(* PLC project HdySimulator Functions library, Porcheson AuxBAse Framework 0.0 *)
(* stored: creationDateTime 2023-02-10T00:00:00, modificationDateTime 2026-02-10T00:00:00 *)

FUNCTION_BLOCK HDY_CreateSimAxis
  VAR_INPUT
    AXISTYPE : USINT;
    MAXVEL : REAL;
    MAXACC : REAL;
    MAXDEC : REAL;
  END_VAR
  VAR_OUTPUT
    AXISID : SINT;
    DONE : BOOL;
  END_VAR

						{{ extern void __mcl_cmd_createSimAxis(HDY_CREATESIMAXIS *data__);	__mcl_cmd_createSimAxis(data__);	 }}	
					
END_FUNCTION_BLOCK

FUNCTION_BLOCK HDY_MoveSimAxis
  VAR_INPUT
    ENABLE : BOOL;
    AXISID : SINT;
    CMD_RPM : REAL;
    DIRECTION : SINT;
  END_VAR
  VAR_OUTPUT
    BUSY : BOOL;
  END_VAR

						{{ extern void __mcl_cmd_moveSimAxis(HDY_MOVESIMAXIS *data__);	__mcl_cmd_moveSimAxis(data__);	 }}	
					
END_FUNCTION_BLOCK

FUNCTION_BLOCK HDY_ReadSimAxis
  VAR_INPUT
    ENABLE : BOOL;
    AXISID : SINT;
  END_VAR
  VAR_OUTPUT
    ACTIVE : BOOL;
    POS_MM : REAL;
    VEL_MM_S : REAL;
    PRESSURE_BAR : REAL;
    BUSY : BOOL;
  END_VAR

						{{ extern void __mcl_cmd_readSimAxis(HDY_READSIMAXIS *data__);	__mcl_cmd_readSimAxis(data__);	 }}	
					
END_FUNCTION_BLOCK
